INTERFACE I_NodeVisitor EXTENDS I_ContentVisitor, I_ParameterVisitor, I_ExtensionVisitor, I_MetadataVisitor, I_ErrorVisitor, I_InputPortVisitor, I_OutputPortVisitor

METHOD VisitNode
VAR_INPUT
	VisitingNode : I_Node;
END_VAR
END_METHOD

END_INTERFACE

(* stored: Version 1.1.0.1, ProductVersion 3.1.4024.12
   Itf I_NodeVisitor: Id {1d67d982-c89b-0cea-2742-6d34a1ca6ed0}
   Method VisitNode: Id {6580424a-37ae-0ba7-1410-7c86db6447b0} *)
